(* PLC project Generated.project, CODESYS CODESYS V3.5 SP19 Patch 1 *)
(* stored: creationDateTime 2026-08-18T01:34:48.440034, modificationDateTime 2026-08-18T01:34:48.440034 *)

(* ═══════════════════════════════════════════════════════════════ ST_CycleCfg — Configuration du cycle semi-automatique SetDepth_M/SetOffset_M protégés par persistance GVL_PERSISTENT ═══════════════════════════════════════════════════════════════ *)
TYPE ST_CycleCfg : STRUCT
  SetDepth_M : REAL := -12.5;  (* 📐 Profondeur de dragage cible (m, négative) *)
  SetOffset_M : REAL := 1.5;  (* 📐 Décalage cible de fermeture de la benne (m) *)
  Initialized : BOOL := FALSE;  (* 🚦 flag restauration boot *)
END_STRUCT;
END_TYPE

(* ======================================================================= 💾 FB_CfgPersistBridge_CycleCfg — Pont persistance pour ST_CycleCfg ─────────────────────────────────────────────────────────────── 🎯 Rôle : Restauration et synchronisation bidirectionnelle IHM / Persist 💾 Persistance : Transfert GVL_PERSISTENT <-> GVL_IHM sur Initialized 📄 Doc métier : DOC/AF/AF_Partie-03_Contrats_Composants_v2.1.md §3 ======================================================================= *)
FUNCTION_BLOCK FB_CfgPersistBridge_CycleCfg
  VAR_OUTPUT
    JustRestored : BOOL;  (* === ETATS RESTAURATION === <-- [STAT] Vrai sur le cycle de restauration initiale *)
  END_VAR
  VAR_IN_OUT
    Hmi : ST_CycleCfg;  (* === BUS CONFIGURATION ET PERSISTANCE === <-> [BUS] Structure de configuration IHM *)
    Persist : ST_CycleCfg;  (* <-> [BUS] Structure de configuration persistante *)
  END_VAR

            

JustRestored := FALSE;
IF NOT Hmi.Initialized THEN
    Hmi := Persist;
    Hmi.Initialized := TRUE;
    JustRestored := TRUE;
ELSE
    Persist := Hmi;
END_IF;

          
END_FUNCTION_BLOCK
